// TIA Portal V20 export
DATA_BLOCK "IdentRfInterfaceHmi"   // DB218
// stored: InstanceOfName typeIdentRfHmi, InstanceOfType UDT
"typeIdentRfHmi"
   // VAR
   //    selectedUnit : USInt := 1;
   //    selectedEM : USInt := 6;
   //    rfReaderId : USInt := 0;
   //    numberOfRf : USInt := 0;
   //    rfReader : Array[0.."NO_OF_RF_IDENT_DEVICES"] of "LSicar_typeIdentInterfaceHmi";
   // END_VAR
BEGIN
   rfReader[0..1].deviceName := WSTRING#'';
   rfReader[0..1].deviceType := WSTRING#'';
   rfReader[0..1].deviceId := 0;
   rfReader[0..1].tagType := WSTRING#'';
   rfReader[0..1].cameraMode := WSTRING#'';
   rfReader[0..1].resultState := WSTRING#'';
   rfReader[0..1].progNo := 0;
   rfReader[0..1].progNumberWrite := 0;
   rfReader[0..1].pushbutton := 16#0000;
   rfReader[0..1].enablePushbutton := 16#0000;
   rfReader[0..1].status := 16#0000;
   rfReader[0..1].alarmCategorie := 0;
   rfReader[0..1].alarmNo := 0;
   rfReader[0..1].alarmCode := 16#0000_0000;
   rfReader[0..1].resultColor := 0;
   rfReader[0..1].statusColorCode := 0;
   rfReader[0..1].datRead1 := '';
   rfReader[0..1].datRead2 := '';
   rfReader[0..1].datRead3 := '';
   rfReader[0..1].datRead4 := '';
   rfReader[0..1].datWrite1 := '';
   rfReader[0..1].datWrite2 := '';
   rfReader[0..1].datWrite3 := '';
   rfReader[0..1].datWrite4 := '';
END_DATA_BLOCK
